# EPICS substitutions: dl205/dl205App/Db/depo-plc-gv.substitutions
file "depo-plc-gv14-calc.template" { pattern
 {Sys, Dev	}
 {Depo, "{GV:1}"}
 {Depo, "{GV:4}"}
}

file "depo-plc-gv23-calc.template" { pattern
 {Sys, Dev	}
 {Depo, "{GV:2}"}
 {Depo, "{GV:3}"}
}
